// TIA Portal V19 export
DATA_BLOCK "PPrfArchive1"   // DB87
// stored: IsOnlyStoredInLoadMemory true, MemoryReserve 0
   VAR RETAIN
      PRG : Array[1.."PPRF_TOTAL_ARCHIVE_ITEMS"] of "PPrf_Data";
   END_VAR
BEGIN
   PRG[1].Header.PrgNo := 1;
   PRG[2].Header.PrgNo := 107;
   PRG[3].Header.PrgNo := 101;
   PRG[4].Header.PrgNo := 102;
   PRG[5].Header.PrgNo := 103;
   PRG[6].Header.PrgNo := 104;
   PRG[7].Header.PrgNo := 110;
   PRG[8].Header.PrgNo := 105;
   PRG[9].Header.PrgNo := 106;
   PRG[10].Header.PrgNo := 108;
   PRG[11].Header.PrgNo := 109;
   PRG[12].Header.PrgNo := 111;
   PRG[13].Header.PrgNo := 112;
   PRG[14].Header.PrgNo := 201;
   PRG[15].Header.PrgNo := 202;
   PRG[16].Header.PrgNo := 203;
   PRG[17].Header.PrgNo := 204;
   PRG[18].Header.PrgNo := 205;
   PRG[19].Header.PrgNo := 206;
   PRG[20].Header.PrgNo := 207;
   PRG[21].Header.PrgNo := 208;
   PRG[22].Header.PrgNo := 209;
   PRG[23].Header.PrgNo := 210;
   PRG[24].Header.PrgNo := 211;
   PRG[25].Header.PrgNo := 212;
   PRG[1].Header.PrgName := 'TEST';
   PRG[2].Header.PrgName := 'Semigusci G12L <S120x45x1.25>';
   PRG[3].Header.PrgName := 'Semigusci G06L <S060x40x1.25>';
   PRG[4].Header.PrgName := 'Semigusci G07L <S070x40x1.25>';
   PRG[5].Header.PrgName := 'Semigusci G08L <S080x40x1.25>';
   PRG[6].Header.PrgName := 'Semigusci G09L <S090x40x1.25>';
   PRG[7].Header.PrgName := 'Semigusci G14N <S140x45x1.5>';
   PRG[8].Header.PrgName := 'Semigusci G10L <S100x40x1.25>';
   PRG[9].Header.PrgName := 'Semigusci G11L <S110x45x1.25>';
   PRG[10].Header.PrgName := 'Semigusci G13L <S130x45x1.25>';
   PRG[11].Header.PrgName := 'Semigusci G14L <S140x45x1.25>';
   PRG[12].Header.PrgName := 'Semigusci G15N <S150x45x1.5>';
   PRG[13].Header.PrgName := 'Semigusci G18N <S180x45x1.5>';
   PRG[14].Header.PrgName := 'Accoppiato G06L <C060x40x1.25>';
   PRG[15].Header.PrgName := 'Accoppiato G07L <C070x40x1.25>';
   PRG[16].Header.PrgName := 'Accoppiato G08L <C080x40x1.25>';
   PRG[17].Header.PrgName := 'Accoppiato G09L <C090x40x1.25>';
   PRG[18].Header.PrgName := 'Accoppiato G10L <C100x40x1.25>';
   PRG[19].Header.PrgName := 'Accoppiato G11L <C110x45x1.25>';
   PRG[20].Header.PrgName := 'Accoppiato G12L <C120x45x1.25>';
   PRG[21].Header.PrgName := 'Accoppiato G13L <C130x45x1.25>';
   PRG[22].Header.PrgName := 'Accoppiato G14L <C140x45x1.25>';
   PRG[23].Header.PrgName := 'Accoppiato G14N <C140x45x1.5>';
   PRG[24].Header.PrgName := 'Accoppiato G15N <C150x45x1.5>';
   PRG[25].Header.PrgName := 'Accoppiato G18N <C180x45x1.5>';
   PRG[1..2].GeneralData.Material_Width := 220.0;
   PRG[3].GeneralData.Material_Width := 149.0;
   PRG[4].GeneralData.Material_Width := 159.0;
   PRG[5].GeneralData.Material_Width := 169.0;
   PRG[6].GeneralData.Material_Width := 179.0;
   PRG[7].GeneralData.Material_Width := 240.0;
   PRG[8].GeneralData.Material_Width := 189.0;
   PRG[9].GeneralData.Material_Width := 210.0;
   PRG[10].GeneralData.Material_Width := 230.0;
   PRG[11].GeneralData.Material_Width := 240.0;
   PRG[12].GeneralData.Material_Width := 255.0;
   PRG[13].GeneralData.Material_Width := 280.0;
   PRG[14].GeneralData.Material_Width := 149.0;
   PRG[15].GeneralData.Material_Width := 159.0;
   PRG[16].GeneralData.Material_Width := 169.0;
   PRG[17].GeneralData.Material_Width := 179.0;
   PRG[18].GeneralData.Material_Width := 189.0;
   PRG[19].GeneralData.Material_Width := 210.0;
   PRG[20].GeneralData.Material_Width := 220.0;
   PRG[21].GeneralData.Material_Width := 230.0;
   PRG[22..23].GeneralData.Material_Width := 240.0;
   PRG[24].GeneralData.Material_Width := 255.0;
   PRG[25].GeneralData.Material_Width := 280.0;
   PRG[26].GeneralData.Material_Width := 0.0;
   PRG[27].GeneralData.Material_Width := 214.0;
   PRG[28].GeneralData.Material_Width := 0.0;
   PRG[29].GeneralData.Material_Width := 236.0;
   PRG[30].GeneralData.Material_Width := 208.0;
   PRG[1].GeneralData.Material_Thickness := 0.0;
   PRG[3].GeneralData.Material_Thickness := 0.0;
   PRG[6..26].GeneralData.Material_Thickness := 0.0;
   PRG[27].GeneralData.Material_Thickness := 2.0;
   PRG[28].GeneralData.Material_Thickness := 0.0;
   PRG[29].GeneralData.Material_Thickness := 3.0;
   PRG[30].GeneralData.Material_Thickness := 1.5;
   PRG[1..25].GeneralData.Material_Tol_Min := -0.5;
   PRG[1..25].GeneralData.Material_Tol_Max := 0.5;
   PRG[14..25].GeneralData.Beam_Code := 1;
   PRG[1].GeneralData.Beam_W_A_Code := 40;
   PRG[2].GeneralData.Beam_W_A_Code := 45;
   PRG[3..6].GeneralData.Beam_W_A_Code := 40;
   PRG[7].GeneralData.Beam_W_A_Code := 45;
   PRG[8].GeneralData.Beam_W_A_Code := 40;
   PRG[9..13].GeneralData.Beam_W_A_Code := 45;
   PRG[14..18].GeneralData.Beam_W_A_Code := 40;
   PRG[19..25].GeneralData.Beam_W_A_Code := 45;
   PRG[1].GeneralData.Beam_H_B_Code := 60;
   PRG[2].GeneralData.Beam_H_B_Code := 120;
   PRG[3].GeneralData.Beam_H_B_Code := 60;
   PRG[4].GeneralData.Beam_H_B_Code := 70;
   PRG[5].GeneralData.Beam_H_B_Code := 80;
   PRG[6].GeneralData.Beam_H_B_Code := 90;
   PRG[7].GeneralData.Beam_H_B_Code := 140;
   PRG[8].GeneralData.Beam_H_B_Code := 100;
   PRG[9].GeneralData.Beam_H_B_Code := 110;
   PRG[10].GeneralData.Beam_H_B_Code := 130;
   PRG[11].GeneralData.Beam_H_B_Code := 140;
   PRG[12].GeneralData.Beam_H_B_Code := 150;
   PRG[13].GeneralData.Beam_H_B_Code := 180;
   PRG[14].GeneralData.Beam_H_B_Code := 60;
   PRG[15].GeneralData.Beam_H_B_Code := 70;
   PRG[16].GeneralData.Beam_H_B_Code := 80;
   PRG[17].GeneralData.Beam_H_B_Code := 90;
   PRG[18].GeneralData.Beam_H_B_Code := 100;
   PRG[19].GeneralData.Beam_H_B_Code := 110;
   PRG[20].GeneralData.Beam_H_B_Code := 120;
   PRG[21].GeneralData.Beam_H_B_Code := 130;
   PRG[22..23].GeneralData.Beam_H_B_Code := 140;
   PRG[24].GeneralData.Beam_H_B_Code := 150;
   PRG[25].GeneralData.Beam_H_B_Code := 180;
   PRG[1..6].GeneralData.Beam_TK_Code := 125;
   PRG[7].GeneralData.Beam_TK_Code := 150;
   PRG[8..11].GeneralData.Beam_TK_Code := 125;
   PRG[12..13].GeneralData.Beam_TK_Code := 150;
   PRG[14..22].GeneralData.Beam_TK_Code := 125;
   PRG[23..25].GeneralData.Beam_TK_Code := 150;
   PRG[1..25].GeneralData.Beam_Len_Tol_Min := -1.0;
   PRG[4..25].GeneralData.Thickness_Mark := 1;
   PRG[4..25].GeneralData.Trace_Mark := 1;
   PRG[1..2].GeneralData.PackLayout_BeamsPerLayer := 10;
   PRG[3..13].GeneralData.PackLayout_BeamsPerLayer := 0;
   PRG[14].GeneralData.PackLayout_BeamsPerLayer := 9;
   PRG[15].GeneralData.PackLayout_BeamsPerLayer := 8;
   PRG[16].GeneralData.PackLayout_BeamsPerLayer := 7;
   PRG[17..18].GeneralData.PackLayout_BeamsPerLayer := 6;
   PRG[19].GeneralData.PackLayout_BeamsPerLayer := 55;
   PRG[20].GeneralData.PackLayout_BeamsPerLayer := 5;
   PRG[21..24].GeneralData.PackLayout_BeamsPerLayer := 4;
   PRG[25].GeneralData.PackLayout_BeamsPerLayer := 3;
   PRG[1..2].GeneralData.PackLayout_Layers_Qty := 5;
   PRG[3..13].GeneralData.PackLayout_Layers_Qty := 0;
   PRG[14..25].GeneralData.PackLayout_Layers_Qty := 11;
   PRG[2].SetUp.Aut.Rollformer.Passaggio02_OP := 1.1;
   PRG[3..6].SetUp.Aut.Rollformer.Passaggio02_OP := 5.0;
   PRG[7].SetUp.Aut.Rollformer.Passaggio02_OP := 0.8;
   PRG[8].SetUp.Aut.Rollformer.Passaggio02_OP := 5.0;
   PRG[9..11].SetUp.Aut.Rollformer.Passaggio02_OP := 1.25;
   PRG[12..13].SetUp.Aut.Rollformer.Passaggio02_OP := 1.5;
   PRG[14..18].SetUp.Aut.Rollformer.Passaggio02_OP := 5.0;
   PRG[19].SetUp.Aut.Rollformer.Passaggio02_OP := 1.25;
   PRG[20].SetUp.Aut.Rollformer.Passaggio02_OP := 0.9137398;
   PRG[21].SetUp.Aut.Rollformer.Passaggio02_OP := 1.25;
   PRG[22].SetUp.Aut.Rollformer.Passaggio02_OP := 0.6;
   PRG[23].SetUp.Aut.Rollformer.Passaggio02_OP := 1.0;
   PRG[24].SetUp.Aut.Rollformer.Passaggio02_OP := 1.5;
   PRG[25].SetUp.Aut.Rollformer.Passaggio02_OP := 0.8;
   PRG[2].SetUp.Aut.Rollformer.Passaggio02_MOT := 1.1;
   PRG[3..6].SetUp.Aut.Rollformer.Passaggio02_MOT := 5.0;
   PRG[7].SetUp.Aut.Rollformer.Passaggio02_MOT := 0.8;
   PRG[8].SetUp.Aut.Rollformer.Passaggio02_MOT := 5.0;
   PRG[9..11].SetUp.Aut.Rollformer.Passaggio02_MOT := 1.25;
   PRG[12..13].SetUp.Aut.Rollformer.Passaggio02_MOT := 1.5;
   PRG[14..18].SetUp.Aut.Rollformer.Passaggio02_MOT := 5.0;
   PRG[19].SetUp.Aut.Rollformer.Passaggio02_MOT := 1.25;
   PRG[20].SetUp.Aut.Rollformer.Passaggio02_MOT := 0.9132179;
   PRG[21].SetUp.Aut.Rollformer.Passaggio02_MOT := 1.25;
   PRG[22].SetUp.Aut.Rollformer.Passaggio02_MOT := 0.6;
   PRG[23].SetUp.Aut.Rollformer.Passaggio02_MOT := 1.0;
   PRG[24].SetUp.Aut.Rollformer.Passaggio02_MOT := 1.5;
   PRG[25].SetUp.Aut.Rollformer.Passaggio02_MOT := 0.8;
   PRG[2].SetUp.Aut.Rollformer.Passaggio17_OP := 0.6;
   PRG[3..6].SetUp.Aut.Rollformer.Passaggio17_OP := 1.25;
   PRG[7].SetUp.Aut.Rollformer.Passaggio17_OP := 1.2;
   PRG[8..11].SetUp.Aut.Rollformer.Passaggio17_OP := 1.25;
   PRG[12..13].SetUp.Aut.Rollformer.Passaggio17_OP := 1.5;
   PRG[14..19].SetUp.Aut.Rollformer.Passaggio17_OP := 1.25;
   PRG[20].SetUp.Aut.Rollformer.Passaggio17_OP := 0.4124924;
   PRG[21].SetUp.Aut.Rollformer.Passaggio17_OP := 1.25;
   PRG[22].SetUp.Aut.Rollformer.Passaggio17_OP := 0.55;
   PRG[23].SetUp.Aut.Rollformer.Passaggio17_OP := 1.2;
   PRG[24].SetUp.Aut.Rollformer.Passaggio17_OP := 1.5;
   PRG[25].SetUp.Aut.Rollformer.Passaggio17_OP := 1.2;
   PRG[2].SetUp.Aut.Rollformer.Passaggio17_MOT := 0.6;
   PRG[3..6].SetUp.Aut.Rollformer.Passaggio17_MOT := 1.25;
   PRG[7].SetUp.Aut.Rollformer.Passaggio17_MOT := 1.2;
   PRG[8..11].SetUp.Aut.Rollformer.Passaggio17_MOT := 1.25;
   PRG[12..13].SetUp.Aut.Rollformer.Passaggio17_MOT := 1.5;
   PRG[14..19].SetUp.Aut.Rollformer.Passaggio17_MOT := 1.25;
   PRG[20].SetUp.Aut.Rollformer.Passaggio17_MOT := 0.9078614;
   PRG[21].SetUp.Aut.Rollformer.Passaggio17_MOT := 1.25;
   PRG[22].SetUp.Aut.Rollformer.Passaggio17_MOT := 0.55;
   PRG[23].SetUp.Aut.Rollformer.Passaggio17_MOT := 1.2;
   PRG[24].SetUp.Aut.Rollformer.Passaggio17_MOT := 1.5;
   PRG[25].SetUp.Aut.Rollformer.Passaggio17_MOT := 1.2;
   PRG[2].SetUp.Aut.Rollformer.Passaggio18_OP := 1.4;
   PRG[3..6].SetUp.Aut.Rollformer.Passaggio18_OP := 1.25;
   PRG[7].SetUp.Aut.Rollformer.Passaggio18_OP := 1.1;
   PRG[8..11].SetUp.Aut.Rollformer.Passaggio18_OP := 1.25;
   PRG[12..13].SetUp.Aut.Rollformer.Passaggio18_OP := 1.5;
   PRG[14..19].SetUp.Aut.Rollformer.Passaggio18_OP := 1.25;
   PRG[20].SetUp.Aut.Rollformer.Passaggio18_OP := 1.405658;
   PRG[21].SetUp.Aut.Rollformer.Passaggio18_OP := 1.25;
   PRG[22].SetUp.Aut.Rollformer.Passaggio18_OP := 1.4;
   PRG[23].SetUp.Aut.Rollformer.Passaggio18_OP := 1.1;
   PRG[24].SetUp.Aut.Rollformer.Passaggio18_OP := 1.5;
   PRG[25].SetUp.Aut.Rollformer.Passaggio18_OP := 1.1;
   PRG[2].SetUp.Aut.Rollformer.Passaggio18_MOT := 1.4;
   PRG[3..6].SetUp.Aut.Rollformer.Passaggio18_MOT := 1.25;
   PRG[7].SetUp.Aut.Rollformer.Passaggio18_MOT := 1.1;
   PRG[8..11].SetUp.Aut.Rollformer.Passaggio18_MOT := 1.25;
   PRG[12..13].SetUp.Aut.Rollformer.Passaggio18_MOT := 1.5;
   PRG[14..19].SetUp.Aut.Rollformer.Passaggio18_MOT := 1.25;
   PRG[20].SetUp.Aut.Rollformer.Passaggio18_MOT := 1.407493;
   PRG[21].SetUp.Aut.Rollformer.Passaggio18_MOT := 1.25;
   PRG[22].SetUp.Aut.Rollformer.Passaggio18_MOT := 1.4;
   PRG[23].SetUp.Aut.Rollformer.Passaggio18_MOT := 1.1;
   PRG[24].SetUp.Aut.Rollformer.Passaggio18_MOT := 1.5;
   PRG[25].SetUp.Aut.Rollformer.Passaggio18_MOT := 1.1;
   PRG[2].SetUp.Aut.Rollformer.Cassetta_1_OP := 101.75;
   PRG[3].SetUp.Aut.Rollformer.Cassetta_1_OP := 71.1;
   PRG[4].SetUp.Aut.Rollformer.Cassetta_1_OP := 76.1;
   PRG[5].SetUp.Aut.Rollformer.Cassetta_1_OP := 81.1;
   PRG[6].SetUp.Aut.Rollformer.Cassetta_1_OP := 86.1;
   PRG[7].SetUp.Aut.Rollformer.Cassetta_1_OP := 112.4;
   PRG[8].SetUp.Aut.Rollformer.Cassetta_1_OP := 91.1;
   PRG[9].SetUp.Aut.Rollformer.Cassetta_1_OP := 101.1;
   PRG[10].SetUp.Aut.Rollformer.Cassetta_1_OP := 111.1;
   PRG[11].SetUp.Aut.Rollformer.Cassetta_1_OP := 116.1;
   PRG[12].SetUp.Aut.Rollformer.Cassetta_1_OP := 120.0;
   PRG[13].SetUp.Aut.Rollformer.Cassetta_1_OP := 135.0;
   PRG[14].SetUp.Aut.Rollformer.Cassetta_1_OP := 71.1;
   PRG[15].SetUp.Aut.Rollformer.Cassetta_1_OP := 76.1;
   PRG[16].SetUp.Aut.Rollformer.Cassetta_1_OP := 81.1;
   PRG[17].SetUp.Aut.Rollformer.Cassetta_1_OP := 86.1;
   PRG[18].SetUp.Aut.Rollformer.Cassetta_1_OP := 91.1;
   PRG[19].SetUp.Aut.Rollformer.Cassetta_1_OP := 101.1;
   PRG[20].SetUp.Aut.Rollformer.Cassetta_1_OP := 101.7414;
   PRG[21].SetUp.Aut.Rollformer.Cassetta_1_OP := 111.1;
   PRG[22].SetUp.Aut.Rollformer.Cassetta_1_OP := 111.75;
   PRG[23].SetUp.Aut.Rollformer.Cassetta_1_OP := 112.4;
   PRG[24].SetUp.Aut.Rollformer.Cassetta_1_OP := 120.0;
   PRG[25].SetUp.Aut.Rollformer.Cassetta_1_OP := 132.4;
   PRG[2].SetUp.Aut.Rollformer.Cassetta_1_MOT := 105.5;
   PRG[3].SetUp.Aut.Rollformer.Cassetta_1_MOT := 71.2;
   PRG[4].SetUp.Aut.Rollformer.Cassetta_1_MOT := 76.2;
   PRG[5].SetUp.Aut.Rollformer.Cassetta_1_MOT := 81.2;
   PRG[6].SetUp.Aut.Rollformer.Cassetta_1_MOT := 86.2;
   PRG[7].SetUp.Aut.Rollformer.Cassetta_1_MOT := 112.1;
   PRG[8].SetUp.Aut.Rollformer.Cassetta_1_MOT := 91.2;
   PRG[9].SetUp.Aut.Rollformer.Cassetta_1_MOT := 101.2;
   PRG[10].SetUp.Aut.Rollformer.Cassetta_1_MOT := 111.2;
   PRG[11].SetUp.Aut.Rollformer.Cassetta_1_MOT := 116.2;
   PRG[12].SetUp.Aut.Rollformer.Cassetta_1_MOT := 120.0;
   PRG[13].SetUp.Aut.Rollformer.Cassetta_1_MOT := 135.0;
   PRG[14].SetUp.Aut.Rollformer.Cassetta_1_MOT := 71.2;
   PRG[15].SetUp.Aut.Rollformer.Cassetta_1_MOT := 76.2;
   PRG[16].SetUp.Aut.Rollformer.Cassetta_1_MOT := 81.2;
   PRG[17].SetUp.Aut.Rollformer.Cassetta_1_MOT := 86.2;
   PRG[18].SetUp.Aut.Rollformer.Cassetta_1_MOT := 91.2;
   PRG[19].SetUp.Aut.Rollformer.Cassetta_1_MOT := 101.2;
   PRG[20].SetUp.Aut.Rollformer.Cassetta_1_MOT := 106.4;
   PRG[21].SetUp.Aut.Rollformer.Cassetta_1_MOT := 111.2;
   PRG[22].SetUp.Aut.Rollformer.Cassetta_1_MOT := 115.8;
   PRG[23].SetUp.Aut.Rollformer.Cassetta_1_MOT := 112.1;
   PRG[24].SetUp.Aut.Rollformer.Cassetta_1_MOT := 120.0;
   PRG[25].SetUp.Aut.Rollformer.Cassetta_1_MOT := 132.1;
   PRG[2].SetUp.Aut.Rollformer.Cassetta_2_OP := 60.5;
   PRG[3].SetUp.Aut.Rollformer.Cassetta_2_OP := 30.0;
   PRG[4].SetUp.Aut.Rollformer.Cassetta_2_OP := 35.0;
   PRG[5].SetUp.Aut.Rollformer.Cassetta_2_OP := 40.0;
   PRG[6].SetUp.Aut.Rollformer.Cassetta_2_OP := 45.0;
   PRG[7].SetUp.Aut.Rollformer.Cassetta_2_OP := 70.1;
   PRG[8].SetUp.Aut.Rollformer.Cassetta_2_OP := 50.0;
   PRG[9].SetUp.Aut.Rollformer.Cassetta_2_OP := 55.0;
   PRG[10].SetUp.Aut.Rollformer.Cassetta_2_OP := 65.0;
   PRG[11].SetUp.Aut.Rollformer.Cassetta_2_OP := 70.0;
   PRG[12].SetUp.Aut.Rollformer.Cassetta_2_OP := 75.0;
   PRG[13].SetUp.Aut.Rollformer.Cassetta_2_OP := 90.0;
   PRG[14].SetUp.Aut.Rollformer.Cassetta_2_OP := 30.0;
   PRG[15].SetUp.Aut.Rollformer.Cassetta_2_OP := 35.0;
   PRG[16].SetUp.Aut.Rollformer.Cassetta_2_OP := 40.0;
   PRG[17].SetUp.Aut.Rollformer.Cassetta_2_OP := 45.0;
   PRG[18].SetUp.Aut.Rollformer.Cassetta_2_OP := 50.0;
   PRG[19].SetUp.Aut.Rollformer.Cassetta_2_OP := 55.0;
   PRG[20].SetUp.Aut.Rollformer.Cassetta_2_OP := 60.5;
   PRG[21].SetUp.Aut.Rollformer.Cassetta_2_OP := 65.0;
   PRG[22].SetUp.Aut.Rollformer.Cassetta_2_OP := 70.5;
   PRG[23].SetUp.Aut.Rollformer.Cassetta_2_OP := 69.9;
   PRG[24].SetUp.Aut.Rollformer.Cassetta_2_OP := 75.0;
   PRG[25].SetUp.Aut.Rollformer.Cassetta_2_OP := 90.1;
   PRG[2].SetUp.Aut.Rollformer.Cassetta_2_MOT := 60.35;
   PRG[3].SetUp.Aut.Rollformer.Cassetta_2_MOT := 30.25;
   PRG[4].SetUp.Aut.Rollformer.Cassetta_2_MOT := 35.25;
   PRG[5].SetUp.Aut.Rollformer.Cassetta_2_MOT := 40.25;
   PRG[6].SetUp.Aut.Rollformer.Cassetta_2_MOT := 45.25;
   PRG[7].SetUp.Aut.Rollformer.Cassetta_2_MOT := 70.5;
   PRG[8].SetUp.Aut.Rollformer.Cassetta_2_MOT := 50.25;
   PRG[9].SetUp.Aut.Rollformer.Cassetta_2_MOT := 55.25;
   PRG[10].SetUp.Aut.Rollformer.Cassetta_2_MOT := 65.25;
   PRG[11].SetUp.Aut.Rollformer.Cassetta_2_MOT := 70.25;
   PRG[12].SetUp.Aut.Rollformer.Cassetta_2_MOT := 75.0;
   PRG[13].SetUp.Aut.Rollformer.Cassetta_2_MOT := 90.0;
   PRG[14].SetUp.Aut.Rollformer.Cassetta_2_MOT := 30.25;
   PRG[15].SetUp.Aut.Rollformer.Cassetta_2_MOT := 35.25;
   PRG[16].SetUp.Aut.Rollformer.Cassetta_2_MOT := 40.25;
   PRG[17].SetUp.Aut.Rollformer.Cassetta_2_MOT := 45.25;
   PRG[18].SetUp.Aut.Rollformer.Cassetta_2_MOT := 50.25;
   PRG[19].SetUp.Aut.Rollformer.Cassetta_2_MOT := 55.25;
   PRG[20].SetUp.Aut.Rollformer.Cassetta_2_MOT := 60.00948;
   PRG[21].SetUp.Aut.Rollformer.Cassetta_2_MOT := 65.25;
   PRG[22..23].SetUp.Aut.Rollformer.Cassetta_2_MOT := 70.3;
   PRG[24].SetUp.Aut.Rollformer.Cassetta_2_MOT := 75.0;
   PRG[25].SetUp.Aut.Rollformer.Cassetta_2_MOT := 90.5;
   PRG[2].SetUp.Aut.Rollformer.Cassetta_3_OP := 59.75;
   PRG[3].SetUp.Aut.Rollformer.Cassetta_3_OP := 30.0;
   PRG[4].SetUp.Aut.Rollformer.Cassetta_3_OP := 35.0;
   PRG[5].SetUp.Aut.Rollformer.Cassetta_3_OP := 40.0;
   PRG[6].SetUp.Aut.Rollformer.Cassetta_3_OP := 45.0;
   PRG[7].SetUp.Aut.Rollformer.Cassetta_3_OP := 70.1;
   PRG[8].SetUp.Aut.Rollformer.Cassetta_3_OP := 50.0;
   PRG[9].SetUp.Aut.Rollformer.Cassetta_3_OP := 55.0;
   PRG[10].SetUp.Aut.Rollformer.Cassetta_3_OP := 65.0;
   PRG[11].SetUp.Aut.Rollformer.Cassetta_3_OP := 70.0;
   PRG[12].SetUp.Aut.Rollformer.Cassetta_3_OP := 75.0;
   PRG[13].SetUp.Aut.Rollformer.Cassetta_3_OP := 90.0;
   PRG[14].SetUp.Aut.Rollformer.Cassetta_3_OP := 30.0;
   PRG[15].SetUp.Aut.Rollformer.Cassetta_3_OP := 35.0;
   PRG[16].SetUp.Aut.Rollformer.Cassetta_3_OP := 40.0;
   PRG[17].SetUp.Aut.Rollformer.Cassetta_3_OP := 45.0;
   PRG[18].SetUp.Aut.Rollformer.Cassetta_3_OP := 50.0;
   PRG[19].SetUp.Aut.Rollformer.Cassetta_3_OP := 55.0;
   PRG[20].SetUp.Aut.Rollformer.Cassetta_3_OP := 59.74569;
   PRG[21].SetUp.Aut.Rollformer.Cassetta_3_OP := 65.0;
   PRG[22].SetUp.Aut.Rollformer.Cassetta_3_OP := 70.5;
   PRG[23].SetUp.Aut.Rollformer.Cassetta_3_OP := 69.9;
   PRG[24].SetUp.Aut.Rollformer.Cassetta_3_OP := 75.0;
   PRG[25].SetUp.Aut.Rollformer.Cassetta_3_OP := 90.1;
   PRG[2].SetUp.Aut.Rollformer.Cassetta_3_MOT := 60.5;
   PRG[3].SetUp.Aut.Rollformer.Cassetta_3_MOT := 30.25;
   PRG[4].SetUp.Aut.Rollformer.Cassetta_3_MOT := 35.25;
   PRG[5].SetUp.Aut.Rollformer.Cassetta_3_MOT := 40.25;
   PRG[6].SetUp.Aut.Rollformer.Cassetta_3_MOT := 45.25;
   PRG[7].SetUp.Aut.Rollformer.Cassetta_3_MOT := 70.5;
   PRG[8].SetUp.Aut.Rollformer.Cassetta_3_MOT := 50.25;
   PRG[9].SetUp.Aut.Rollformer.Cassetta_3_MOT := 55.25;
   PRG[10].SetUp.Aut.Rollformer.Cassetta_3_MOT := 65.25;
   PRG[11].SetUp.Aut.Rollformer.Cassetta_3_MOT := 70.25;
   PRG[12].SetUp.Aut.Rollformer.Cassetta_3_MOT := 75.0;
   PRG[13].SetUp.Aut.Rollformer.Cassetta_3_MOT := 90.0;
   PRG[14].SetUp.Aut.Rollformer.Cassetta_3_MOT := 30.25;
   PRG[15].SetUp.Aut.Rollformer.Cassetta_3_MOT := 35.25;
   PRG[16].SetUp.Aut.Rollformer.Cassetta_3_MOT := 40.25;
   PRG[17].SetUp.Aut.Rollformer.Cassetta_3_MOT := 45.25;
   PRG[18].SetUp.Aut.Rollformer.Cassetta_3_MOT := 50.25;
   PRG[19].SetUp.Aut.Rollformer.Cassetta_3_MOT := 55.25;
   PRG[20].SetUp.Aut.Rollformer.Cassetta_3_MOT := 60.00629;
   PRG[21].SetUp.Aut.Rollformer.Cassetta_3_MOT := 65.25;
   PRG[22..23].SetUp.Aut.Rollformer.Cassetta_3_MOT := 70.3;
   PRG[24].SetUp.Aut.Rollformer.Cassetta_3_MOT := 75.0;
   PRG[25].SetUp.Aut.Rollformer.Cassetta_3_MOT := 90.5;
   PRG[2].SetUp.Aut.Bordatrice.Passaggio01_L := 45.0;
   PRG[5..7].SetUp.Aut.Bordatrice.Passaggio01_L := 45.0;
   PRG[20].SetUp.Aut.Bordatrice.Passaggio01_L := 46.09322;
   PRG[22].SetUp.Aut.Bordatrice.Passaggio01_L := 46.0;
   PRG[23..24].SetUp.Aut.Bordatrice.Passaggio01_L := 45.0;
   PRG[25].SetUp.Aut.Bordatrice.Passaggio01_L := 45.5;
   PRG[2].SetUp.Aut.Bordatrice.Passaggio01_R := 45.0;
   PRG[5..7].SetUp.Aut.Bordatrice.Passaggio01_R := 45.0;
   PRG[20].SetUp.Aut.Bordatrice.Passaggio01_R := 46.09262;
   PRG[22].SetUp.Aut.Bordatrice.Passaggio01_R := 46.0;
   PRG[23..24].SetUp.Aut.Bordatrice.Passaggio01_R := 45.0;
   PRG[25].SetUp.Aut.Bordatrice.Passaggio01_R := 45.5;
   PRG[2].SetUp.Aut.Bordatrice.Passaggio02_L := 45.0;
   PRG[6].SetUp.Aut.Bordatrice.Passaggio02_L := 45.0;
   PRG[7].SetUp.Aut.Bordatrice.Passaggio02_L := 44.85;
   PRG[20].SetUp.Aut.Bordatrice.Passaggio02_L := 45.00256;
   PRG[22].SetUp.Aut.Bordatrice.Passaggio02_L := 45.0;
   PRG[23].SetUp.Aut.Bordatrice.Passaggio02_L := 44.8;
   PRG[24].SetUp.Aut.Bordatrice.Passaggio02_L := 45.0;
   PRG[25].SetUp.Aut.Bordatrice.Passaggio02_L := 44.5;
   PRG[2].SetUp.Aut.Bordatrice.Passaggio02_R := 45.0;
   PRG[6].SetUp.Aut.Bordatrice.Passaggio02_R := 45.0;
   PRG[7].SetUp.Aut.Bordatrice.Passaggio02_R := 44.85;
   PRG[20].SetUp.Aut.Bordatrice.Passaggio02_R := 45.00402;
   PRG[22].SetUp.Aut.Bordatrice.Passaggio02_R := 45.0;
   PRG[23].SetUp.Aut.Bordatrice.Passaggio02_R := 44.8;
   PRG[24].SetUp.Aut.Bordatrice.Passaggio02_R := 45.0;
   PRG[25].SetUp.Aut.Bordatrice.Passaggio02_R := 44.5;
   PRG[2].SetUp.Aut.Bordatrice.Passaggio03_L := 45.0;
   PRG[6].SetUp.Aut.Bordatrice.Passaggio03_L := 45.0;
   PRG[7].SetUp.Aut.Bordatrice.Passaggio03_L := 43.7;
   PRG[20].SetUp.Aut.Bordatrice.Passaggio03_L := 44.10418;
   PRG[22].SetUp.Aut.Bordatrice.Passaggio03_L := 45.0;
   PRG[23].SetUp.Aut.Bordatrice.Passaggio03_L := 44.0;
   PRG[24].SetUp.Aut.Bordatrice.Passaggio03_L := 45.0;
   PRG[25].SetUp.Aut.Bordatrice.Passaggio03_L := 43.7;
   PRG[2].SetUp.Aut.Bordatrice.Passaggio03_R := 45.0;
   PRG[6].SetUp.Aut.Bordatrice.Passaggio03_R := 45.0;
   PRG[7].SetUp.Aut.Bordatrice.Passaggio03_R := 43.7;
   PRG[20].SetUp.Aut.Bordatrice.Passaggio03_R := 44.49652;
   PRG[22].SetUp.Aut.Bordatrice.Passaggio03_R := 45.0;
   PRG[23].SetUp.Aut.Bordatrice.Passaggio03_R := 44.0;
   PRG[24].SetUp.Aut.Bordatrice.Passaggio03_R := 45.0;
   PRG[25].SetUp.Aut.Bordatrice.Passaggio03_R := 43.7;
   PRG[2].SetUp.Aut.Bordatrice.Passaggio04_L := 45.0;
   PRG[6].SetUp.Aut.Bordatrice.Passaggio04_L := 45.0;
   PRG[7].SetUp.Aut.Bordatrice.Passaggio04_L := 44.2;
   PRG[20].SetUp.Aut.Bordatrice.Passaggio04_L := 43.6;
   PRG[22].SetUp.Aut.Bordatrice.Passaggio04_L := 43.7;
   PRG[23].SetUp.Aut.Bordatrice.Passaggio04_L := 43.9;
   PRG[24].SetUp.Aut.Bordatrice.Passaggio04_L := 45.0;
   PRG[25].SetUp.Aut.Bordatrice.Passaggio04_L := 43.55;
   PRG[2].SetUp.Aut.Bordatrice.Passaggio04_R := 45.0;
   PRG[6].SetUp.Aut.Bordatrice.Passaggio04_R := 45.0;
   PRG[7].SetUp.Aut.Bordatrice.Passaggio04_R := 44.2;
   PRG[20].SetUp.Aut.Bordatrice.Passaggio04_R := 43.5;
   PRG[22].SetUp.Aut.Bordatrice.Passaggio04_R := 43.7;
   PRG[23].SetUp.Aut.Bordatrice.Passaggio04_R := 43.9;
   PRG[24].SetUp.Aut.Bordatrice.Passaggio04_R := 45.0;
   PRG[25].SetUp.Aut.Bordatrice.Passaggio04_R := 43.55;
   PRG[7].SetUp.Aut.Bordatrice.Cassetta_1_OP := 141.0;
   PRG[20].SetUp.Aut.Bordatrice.Cassetta_1_OP := 119.8;
   PRG[22].SetUp.Aut.Bordatrice.Cassetta_1_OP := 139.7;
   PRG[23].SetUp.Aut.Bordatrice.Cassetta_1_OP := 140.5;
   PRG[25].SetUp.Aut.Bordatrice.Cassetta_1_OP := 180.1;
   PRG[2].SetUp.Man.X[15] := 109.3;
   PRG[2].SetUp.Man.X[16] := 111.3;
   PRG[2].SetUp.Man.X[17] := 7.6;
   PRG[2].SetUp.Man.X[18] := 9.5;
   PRG[2].SetUp.Man.X[19] := 7.6;
   PRG[2].SetUp.Man.X[20] := 9.5;
   PRG[2].SetUp.Man.X[21] := 45.1;
   PRG[2].SetUp.Man.X[22] := 43.5;
   PRG[2].SetUp.Man.X[23] := 45.1;
   PRG[2].SetUp.Man.X[24] := 43.5;
   PRG[2].SetUp.Man.X[25] := 45.1;
   PRG[2].SetUp.Man.X[26] := 43.5;
   PRG[2].SetUp.Man.X[27] := 0.1;
   PRG[2].SetUp.Man.X[28] := 87.6;
   PRG[2].SetUp.Man.X[29] := 84.8;
   PRG[2].SetUp.Man.X[30] := 58.75;
   PRG[2].SetUp.Man.X[31] := 60.0;
   PRG[2].SetUp.Man.X[32] := 58.75;
   PRG[2].SetUp.Man.X[33] := 60.0;
   PRG[3].SetUp.Man.X[15] := 77.6;
   PRG[3].SetUp.Man.X[16] := 71.9;
   PRG[3].SetUp.Man.X[17] := 8.4;
   PRG[3].SetUp.Man.X[18] := 7.0;
   PRG[3].SetUp.Man.X[19] := 8.4;
   PRG[3].SetUp.Man.X[20] := 7.0;
   PRG[3].SetUp.Man.X[21] := 40.1;
   PRG[3].SetUp.Man.X[22] := 38.5;
   PRG[3].SetUp.Man.X[23] := 40.1;
   PRG[3].SetUp.Man.X[24] := 38.5;
   PRG[3].SetUp.Man.X[25] := 40.1;
   PRG[3].SetUp.Man.X[26] := 38.5;
   PRG[3].SetUp.Man.X[27] := 1.0;
   PRG[3].SetUp.Man.X[28] := 87.0;
   PRG[3].SetUp.Man.X[29] := 84.2;
   PRG[3].SetUp.Man.X[30] := 28.75;
   PRG[3].SetUp.Man.X[31] := 30.0;
   PRG[3].SetUp.Man.X[32] := 28.75;
   PRG[3].SetUp.Man.X[33] := 30.0;
   PRG[4].SetUp.Man.X[15] := 82.5;
   PRG[4].SetUp.Man.X[16] := 79.5;
   PRG[4].SetUp.Man.X[17] := 9.75;
   PRG[4].SetUp.Man.X[18] := 5.8;
   PRG[4].SetUp.Man.X[19] := 9.75;
   PRG[4].SetUp.Man.X[20] := 5.8;
   PRG[4].SetUp.Man.X[21] := 41.1;
   PRG[4].SetUp.Man.X[22] := 41.2;
   PRG[4].SetUp.Man.X[23] := 41.1;
   PRG[4].SetUp.Man.X[24] := 41.2;
   PRG[4].SetUp.Man.X[25] := 41.1;
   PRG[4].SetUp.Man.X[26] := 41.2;
   PRG[4].SetUp.Man.X[27] := -0.4;
   PRG[4].SetUp.Man.X[30] := 35.0;
   PRG[4].SetUp.Man.X[31] := 33.75;
   PRG[4].SetUp.Man.X[32] := 35.0;
   PRG[4].SetUp.Man.X[33] := 33.75;
   PRG[5].SetUp.Man.X[15] := 87.5;
   PRG[5].SetUp.Man.X[16] := 84.5;
   PRG[5].SetUp.Man.X[17] := 9.75;
   PRG[5].SetUp.Man.X[18] := 5.8;
   PRG[5].SetUp.Man.X[19] := 9.75;
   PRG[5].SetUp.Man.X[20] := 5.8;
   PRG[5].SetUp.Man.X[21] := 41.1;
   PRG[5].SetUp.Man.X[22] := 41.2;
   PRG[5].SetUp.Man.X[23] := 41.1;
   PRG[5].SetUp.Man.X[24] := 41.2;
   PRG[5].SetUp.Man.X[25] := 41.1;
   PRG[5].SetUp.Man.X[26] := 41.2;
   PRG[5].SetUp.Man.X[27] := -0.4;
   PRG[5].SetUp.Man.X[30] := 38.75;
   PRG[5].SetUp.Man.X[31] := 40.0;
   PRG[5].SetUp.Man.X[32] := 38.75;
   PRG[5].SetUp.Man.X[33] := 40.0;
   PRG[6].SetUp.Man.X[15] := 92.5;
   PRG[6].SetUp.Man.X[16] := 89.5;
   PRG[6].SetUp.Man.X[17] := 9.75;
   PRG[6].SetUp.Man.X[18] := 5.8;
   PRG[6].SetUp.Man.X[19] := 9.75;
   PRG[6].SetUp.Man.X[20] := 5.8;
   PRG[6].SetUp.Man.X[21] := 41.1;
   PRG[6].SetUp.Man.X[22] := 41.2;
   PRG[6].SetUp.Man.X[23] := 41.1;
   PRG[6].SetUp.Man.X[24] := 41.2;
   PRG[6].SetUp.Man.X[25] := 41.1;
   PRG[6].SetUp.Man.X[26] := 41.2;
   PRG[6].SetUp.Man.X[27] := -0.4;
   PRG[6].SetUp.Man.X[30] := 43.8;
   PRG[6].SetUp.Man.X[31] := 45.0;
   PRG[6].SetUp.Man.X[32] := 43.8;
   PRG[6].SetUp.Man.X[33] := 45.0;
   PRG[7].SetUp.Man.X[15..16] := 122.5;
   PRG[7].SetUp.Man.X[17..20] := 10.0;
   PRG[7].SetUp.Man.X[21..26] := 45.0;
   PRG[7].SetUp.Man.X[30] := 68.5;
   PRG[7].SetUp.Man.X[31] := 70.0;
   PRG[7].SetUp.Man.X[32] := 68.5;
   PRG[7].SetUp.Man.X[33] := 70.0;
   PRG[8].SetUp.Man.X[15] := 97.5;
   PRG[8].SetUp.Man.X[16] := 94.5;
   PRG[8].SetUp.Man.X[17] := 9.75;
   PRG[8].SetUp.Man.X[18] := 5.8;
   PRG[8].SetUp.Man.X[19] := 9.75;
   PRG[8].SetUp.Man.X[20] := 5.8;
   PRG[8].SetUp.Man.X[21] := 41.1;
   PRG[8].SetUp.Man.X[22] := 41.2;
   PRG[8].SetUp.Man.X[23] := 41.1;
   PRG[8].SetUp.Man.X[24] := 41.2;
   PRG[8].SetUp.Man.X[25] := 41.1;
   PRG[8].SetUp.Man.X[26] := 41.2;
   PRG[8].SetUp.Man.X[27] := -0.4;
   PRG[8].SetUp.Man.X[30] := 48.8;
   PRG[8].SetUp.Man.X[31] := 50.0;
   PRG[8].SetUp.Man.X[32] := 48.8;
   PRG[8].SetUp.Man.X[33] := 50.0;
   PRG[9].SetUp.Man.X[15] := 97.5;
   PRG[9].SetUp.Man.X[16] := 94.5;
   PRG[9].SetUp.Man.X[17] := 9.75;
   PRG[9].SetUp.Man.X[18] := 5.8;
   PRG[9].SetUp.Man.X[19] := 9.75;
   PRG[9].SetUp.Man.X[20] := 5.8;
   PRG[9].SetUp.Man.X[21] := 46.1;
   PRG[9].SetUp.Man.X[22] := 46.2;
   PRG[9].SetUp.Man.X[23] := 46.1;
   PRG[9].SetUp.Man.X[24] := 46.2;
   PRG[9].SetUp.Man.X[25] := 46.1;
   PRG[9].SetUp.Man.X[26] := 46.2;
   PRG[9].SetUp.Man.X[27] := -0.4;
   PRG[9].SetUp.Man.X[30] := 53.8;
   PRG[9].SetUp.Man.X[31] := 55.0;
   PRG[9].SetUp.Man.X[32] := 53.8;
   PRG[9].SetUp.Man.X[33] := 55.0;
   PRG[10].SetUp.Man.X[15] := 118.0;
   PRG[10].SetUp.Man.X[16] := 115.0;
   PRG[10].SetUp.Man.X[17] := 9.75;
   PRG[10].SetUp.Man.X[18] := 5.8;
   PRG[10].SetUp.Man.X[19] := 9.8;
   PRG[10].SetUp.Man.X[20] := 5.8;
   PRG[10].SetUp.Man.X[21] := 46.1;
   PRG[10].SetUp.Man.X[22] := 46.2;
   PRG[10].SetUp.Man.X[23] := 46.1;
   PRG[10].SetUp.Man.X[24] := 46.2;
   PRG[10].SetUp.Man.X[25] := 46.1;
   PRG[10].SetUp.Man.X[26] := 46.2;
   PRG[10].SetUp.Man.X[27] := -0.4;
   PRG[10].SetUp.Man.X[30] := 63.75;
   PRG[10].SetUp.Man.X[31] := 65.0;
   PRG[10].SetUp.Man.X[32] := 63.75;
   PRG[10].SetUp.Man.X[33] := 65.0;
   PRG[11].SetUp.Man.X[15] := 123.0;
   PRG[11].SetUp.Man.X[16] := 120.0;
   PRG[11].SetUp.Man.X[17] := 7.6;
   PRG[11].SetUp.Man.X[18] := 9.5;
   PRG[11].SetUp.Man.X[19] := 7.6;
   PRG[11].SetUp.Man.X[20] := 9.5;
   PRG[11].SetUp.Man.X[21] := 46.1;
   PRG[11].SetUp.Man.X[22] := 46.2;
   PRG[11].SetUp.Man.X[23] := 46.1;
   PRG[11].SetUp.Man.X[24] := 46.2;
   PRG[11].SetUp.Man.X[25] := 46.1;
   PRG[11].SetUp.Man.X[26] := 46.2;
   PRG[11].SetUp.Man.X[27] := -0.4;
   PRG[11].SetUp.Man.X[30] := 68.8;
   PRG[11].SetUp.Man.X[31] := 70.0;
   PRG[11].SetUp.Man.X[32] := 68.8;
   PRG[11].SetUp.Man.X[33] := 70.0;
   PRG[12].SetUp.Man.X[15] := 126.5;
   PRG[12].SetUp.Man.X[16] := 124.8;
   PRG[12].SetUp.Man.X[17] := 9.0;
   PRG[12].SetUp.Man.X[18] := 12.25;
   PRG[12].SetUp.Man.X[19] := 9.0;
   PRG[12].SetUp.Man.X[20] := 12.25;
   PRG[12].SetUp.Man.X[21] := 42.5;
   PRG[12].SetUp.Man.X[22] := 42.4;
   PRG[12].SetUp.Man.X[23] := 42.5;
   PRG[12].SetUp.Man.X[24] := 42.4;
   PRG[12].SetUp.Man.X[25] := 42.5;
   PRG[12].SetUp.Man.X[26] := 42.4;
   PRG[12].SetUp.Man.X[27] := 0.1;
   PRG[12].SetUp.Man.X[28] := 86.7;
   PRG[12].SetUp.Man.X[29] := 84.0;
   PRG[12].SetUp.Man.X[30] := 73.5;
   PRG[12].SetUp.Man.X[31] := 75.0;
   PRG[12].SetUp.Man.X[32] := 73.5;
   PRG[12].SetUp.Man.X[33] := 75.0;
   PRG[13].SetUp.Man.X[15..16] := 142.5;
   PRG[13].SetUp.Man.X[17..20] := 10.0;
   PRG[13].SetUp.Man.X[21..26] := 45.0;
   PRG[13].SetUp.Man.X[30] := 88.5;
   PRG[13].SetUp.Man.X[31] := 90.0;
   PRG[13].SetUp.Man.X[32] := 88.5;
   PRG[13].SetUp.Man.X[33] := 90.0;
   PRG[14].SetUp.Man.X[15] := 77.6;
   PRG[14].SetUp.Man.X[16] := 71.9;
   PRG[14].SetUp.Man.X[17] := 8.4;
   PRG[14].SetUp.Man.X[18] := 7.0;
   PRG[14].SetUp.Man.X[19] := 8.4;
   PRG[14].SetUp.Man.X[20] := 7.0;
   PRG[14].SetUp.Man.X[21] := 40.1;
   PRG[14].SetUp.Man.X[22] := 38.5;
   PRG[14].SetUp.Man.X[23] := 40.1;
   PRG[14].SetUp.Man.X[24] := 38.5;
   PRG[14].SetUp.Man.X[25] := 40.1;
   PRG[14].SetUp.Man.X[26] := 38.5;
   PRG[14].SetUp.Man.X[27] := 1.0;
   PRG[14].SetUp.Man.X[28] := 87.0;
   PRG[14].SetUp.Man.X[29] := 84.2;
   PRG[14].SetUp.Man.X[30] := 28.75;
   PRG[14].SetUp.Man.X[31] := 30.0;
   PRG[14].SetUp.Man.X[32] := 28.75;
   PRG[14].SetUp.Man.X[33] := 30.0;
   PRG[15].SetUp.Man.X[15] := 82.5;
   PRG[15].SetUp.Man.X[16] := 79.5;
   PRG[15].SetUp.Man.X[17] := 9.75;
   PRG[15].SetUp.Man.X[18] := 5.8;
   PRG[15].SetUp.Man.X[19] := 9.75;
   PRG[15].SetUp.Man.X[20] := 5.8;
   PRG[15].SetUp.Man.X[21] := 41.1;
   PRG[15].SetUp.Man.X[22] := 41.2;
   PRG[15].SetUp.Man.X[23] := 41.1;
   PRG[15].SetUp.Man.X[24] := 41.2;
   PRG[15].SetUp.Man.X[25] := 41.1;
   PRG[15].SetUp.Man.X[26] := 41.2;
   PRG[15].SetUp.Man.X[27] := -0.4;
   PRG[15].SetUp.Man.X[30] := 35.0;
   PRG[15].SetUp.Man.X[31] := 33.75;
   PRG[15].SetUp.Man.X[32] := 35.0;
   PRG[15].SetUp.Man.X[33] := 33.75;
   PRG[16].SetUp.Man.X[15] := 87.5;
   PRG[16].SetUp.Man.X[16] := 84.5;
   PRG[16].SetUp.Man.X[17] := 9.75;
   PRG[16].SetUp.Man.X[18] := 5.8;
   PRG[16].SetUp.Man.X[19] := 9.75;
   PRG[16].SetUp.Man.X[20] := 5.8;
   PRG[16].SetUp.Man.X[21] := 41.1;
   PRG[16].SetUp.Man.X[22] := 41.2;
   PRG[16].SetUp.Man.X[23] := 41.1;
   PRG[16].SetUp.Man.X[24] := 41.2;
   PRG[16].SetUp.Man.X[25] := 41.1;
   PRG[16].SetUp.Man.X[26] := 41.2;
   PRG[16].SetUp.Man.X[27] := -0.4;
   PRG[16].SetUp.Man.X[30] := 38.75;
   PRG[16].SetUp.Man.X[31] := 40.0;
   PRG[16].SetUp.Man.X[32] := 38.75;
   PRG[16].SetUp.Man.X[33] := 40.0;
   PRG[17].SetUp.Man.X[15] := 92.5;
   PRG[17].SetUp.Man.X[16] := 89.5;
   PRG[17].SetUp.Man.X[17] := 9.75;
   PRG[17].SetUp.Man.X[18] := 5.8;
   PRG[17].SetUp.Man.X[19] := 9.75;
   PRG[17].SetUp.Man.X[20] := 5.8;
   PRG[17].SetUp.Man.X[21] := 41.1;
   PRG[17].SetUp.Man.X[22] := 41.2;
   PRG[17].SetUp.Man.X[23] := 41.1;
   PRG[17].SetUp.Man.X[24] := 41.2;
   PRG[17].SetUp.Man.X[25] := 41.1;
   PRG[17].SetUp.Man.X[26] := 41.2;
   PRG[17].SetUp.Man.X[27] := -0.4;
   PRG[17].SetUp.Man.X[30] := 43.8;
   PRG[17].SetUp.Man.X[31] := 45.0;
   PRG[17].SetUp.Man.X[32] := 43.8;
   PRG[17].SetUp.Man.X[33] := 45.0;
   PRG[18].SetUp.Man.X[15] := 97.5;
   PRG[18].SetUp.Man.X[16] := 94.5;
   PRG[18].SetUp.Man.X[17] := 9.75;
   PRG[18].SetUp.Man.X[18] := 5.8;
   PRG[18].SetUp.Man.X[19] := 9.75;
   PRG[18].SetUp.Man.X[20] := 5.8;
   PRG[18].SetUp.Man.X[21] := 41.1;
   PRG[18].SetUp.Man.X[22] := 41.2;
   PRG[18].SetUp.Man.X[23] := 41.1;
   PRG[18].SetUp.Man.X[24] := 41.2;
   PRG[18].SetUp.Man.X[25] := 41.1;
   PRG[18].SetUp.Man.X[26] := 41.2;
   PRG[18].SetUp.Man.X[27] := -0.4;
   PRG[18].SetUp.Man.X[30] := 48.8;
   PRG[18].SetUp.Man.X[31] := 50.0;
   PRG[18].SetUp.Man.X[32] := 48.8;
   PRG[18].SetUp.Man.X[33] := 50.0;
   PRG[19].SetUp.Man.X[15] := 97.5;
   PRG[19].SetUp.Man.X[16] := 94.5;
   PRG[19].SetUp.Man.X[17] := 9.75;
   PRG[19].SetUp.Man.X[18] := 5.8;
   PRG[19].SetUp.Man.X[19] := 9.75;
   PRG[19].SetUp.Man.X[20] := 5.8;
   PRG[19].SetUp.Man.X[21] := 46.1;
   PRG[19].SetUp.Man.X[22] := 46.2;
   PRG[19].SetUp.Man.X[23] := 46.1;
   PRG[19].SetUp.Man.X[24] := 46.2;
   PRG[19].SetUp.Man.X[25] := 46.1;
   PRG[19].SetUp.Man.X[26] := 46.2;
   PRG[19].SetUp.Man.X[27] := -0.4;
   PRG[19].SetUp.Man.X[30] := 53.8;
   PRG[19].SetUp.Man.X[31] := 55.0;
   PRG[19].SetUp.Man.X[32] := 53.8;
   PRG[19].SetUp.Man.X[33] := 55.0;
   PRG[20].SetUp.Man.X[15] := 109.3;
   PRG[20].SetUp.Man.X[16] := 111.3;
   PRG[20].SetUp.Man.X[17] := 7.6;
   PRG[20].SetUp.Man.X[18] := 9.5;
   PRG[20].SetUp.Man.X[19] := 7.6;
   PRG[20].SetUp.Man.X[20] := 9.5;
   PRG[20].SetUp.Man.X[21] := 45.1;
   PRG[20].SetUp.Man.X[22] := 43.5;
   PRG[20].SetUp.Man.X[23] := 45.1;
   PRG[20].SetUp.Man.X[24] := 43.5;
   PRG[20].SetUp.Man.X[25] := 45.1;
   PRG[20].SetUp.Man.X[26] := 43.5;
   PRG[20].SetUp.Man.X[27] := 0.1;
   PRG[20].SetUp.Man.X[28] := 87.6;
   PRG[20].SetUp.Man.X[29] := 84.8;
   PRG[20].SetUp.Man.X[30] := 58.75;
   PRG[20].SetUp.Man.X[31] := 60.0;
   PRG[20].SetUp.Man.X[32] := 58.75;
   PRG[20].SetUp.Man.X[33] := 60.0;
   PRG[21].SetUp.Man.X[15] := 118.0;
   PRG[21].SetUp.Man.X[16] := 115.0;
   PRG[21].SetUp.Man.X[17] := 9.75;
   PRG[21].SetUp.Man.X[18] := 5.8;
   PRG[21].SetUp.Man.X[19] := 9.8;
   PRG[21].SetUp.Man.X[20] := 5.8;
   PRG[21].SetUp.Man.X[21] := 46.1;
   PRG[21].SetUp.Man.X[22] := 46.2;
   PRG[21].SetUp.Man.X[23] := 46.1;
   PRG[21].SetUp.Man.X[24] := 46.2;
   PRG[21].SetUp.Man.X[25] := 46.1;
   PRG[21].SetUp.Man.X[26] := 46.2;
   PRG[21].SetUp.Man.X[27] := -0.4;
   PRG[21].SetUp.Man.X[30] := 63.75;
   PRG[21].SetUp.Man.X[31] := 65.0;
   PRG[21].SetUp.Man.X[32] := 63.75;
   PRG[21].SetUp.Man.X[33] := 65.0;
   PRG[22].SetUp.Man.X[15] := 123.0;
   PRG[22].SetUp.Man.X[16] := 120.0;
   PRG[22].SetUp.Man.X[17] := 7.6;
   PRG[22].SetUp.Man.X[18] := 9.5;
   PRG[22].SetUp.Man.X[19] := 7.6;
   PRG[22].SetUp.Man.X[20] := 9.5;
   PRG[22].SetUp.Man.X[21] := 46.1;
   PRG[22].SetUp.Man.X[22] := 46.2;
   PRG[22].SetUp.Man.X[23] := 46.1;
   PRG[22].SetUp.Man.X[24] := 46.2;
   PRG[22].SetUp.Man.X[25] := 46.1;
   PRG[22].SetUp.Man.X[26] := 46.2;
   PRG[22].SetUp.Man.X[27] := -0.4;
   PRG[22].SetUp.Man.X[30] := 68.8;
   PRG[22].SetUp.Man.X[31] := 70.0;
   PRG[22].SetUp.Man.X[32] := 68.8;
   PRG[22].SetUp.Man.X[33] := 70.0;
   PRG[23].SetUp.Man.X[15..16] := 122.5;
   PRG[23].SetUp.Man.X[17..20] := 10.0;
   PRG[23].SetUp.Man.X[21..26] := 45.0;
   PRG[23].SetUp.Man.X[30] := 68.5;
   PRG[23].SetUp.Man.X[31] := 70.0;
   PRG[23].SetUp.Man.X[32] := 68.5;
   PRG[23].SetUp.Man.X[33] := 70.0;
   PRG[24].SetUp.Man.X[15] := 126.5;
   PRG[24].SetUp.Man.X[16] := 124.8;
   PRG[24].SetUp.Man.X[17] := 9.0;
   PRG[24].SetUp.Man.X[18] := 12.25;
   PRG[24].SetUp.Man.X[19] := 9.0;
   PRG[24].SetUp.Man.X[20] := 12.25;
   PRG[24].SetUp.Man.X[21] := 42.5;
   PRG[24].SetUp.Man.X[22] := 42.4;
   PRG[24].SetUp.Man.X[23] := 42.5;
   PRG[24].SetUp.Man.X[24] := 42.4;
   PRG[24].SetUp.Man.X[25] := 42.5;
   PRG[24].SetUp.Man.X[26] := 42.4;
   PRG[24].SetUp.Man.X[27] := 0.1;
   PRG[24].SetUp.Man.X[28] := 86.7;
   PRG[24].SetUp.Man.X[29] := 84.0;
   PRG[24].SetUp.Man.X[30] := 73.5;
   PRG[24].SetUp.Man.X[31] := 75.0;
   PRG[24].SetUp.Man.X[32] := 73.5;
   PRG[24].SetUp.Man.X[33] := 75.0;
   PRG[25].SetUp.Man.X[15..16] := 142.5;
   PRG[25].SetUp.Man.X[17..20] := 10.0;
   PRG[25].SetUp.Man.X[21..26] := 45.0;
   PRG[25].SetUp.Man.X[30] := 88.5;
   PRG[25].SetUp.Man.X[31] := 90.0;
   PRG[25].SetUp.Man.X[32] := 88.5;
   PRG[25].SetUp.Man.X[33] := 90.0;
   PRG[2].SetUp.Man.Y[1..2] := 120;
   PRG[3].SetUp.Man.Y[1..2] := 60;
   PRG[4].SetUp.Man.Y[1..2] := 70;
   PRG[5].SetUp.Man.Y[1..2] := 80;
   PRG[6].SetUp.Man.Y[1..2] := 90;
   PRG[7].SetUp.Man.Y[1..2] := 140;
   PRG[8].SetUp.Man.Y[1..2] := 100;
   PRG[9].SetUp.Man.Y[1..2] := 110;
   PRG[10].SetUp.Man.Y[1..2] := 130;
   PRG[11].SetUp.Man.Y[1..2] := 140;
   PRG[12].SetUp.Man.Y[1..2] := 150;
   PRG[13].SetUp.Man.Y[1..2] := 180;
   PRG[14].SetUp.Man.Y[1..2] := 60;
   PRG[15].SetUp.Man.Y[1..2] := 70;
   PRG[16].SetUp.Man.Y[1..2] := 80;
   PRG[17].SetUp.Man.Y[1..2] := 90;
   PRG[18].SetUp.Man.Y[1..2] := 100;
   PRG[19].SetUp.Man.Y[1..2] := 110;
   PRG[20].SetUp.Man.Y[1..2] := 120;
   PRG[21].SetUp.Man.Y[1..2] := 130;
   PRG[22].SetUp.Man.Y[1..2] := 140;
   PRG[23].SetUp.Man.Y[1..2] := 140;
   PRG[24].SetUp.Man.Y[1..2] := 150;
   PRG[25].SetUp.Man.Y[1..2] := 180;
   PRG[1..2].A01_CoilHandling.MaterialFeeding.DecoilerFeedMode := 3;
   PRG[3..25].A01_CoilHandling.MaterialFeeding.DecoilerFeedMode := 1;
   PRG[26].A01_CoilHandling.MaterialFeeding.DecoilerFeedMode := 0;
   PRG[27].A01_CoilHandling.MaterialFeeding.DecoilerFeedMode := 1;
   PRG[28].A01_CoilHandling.MaterialFeeding.DecoilerFeedMode := 0;
   PRG[29..30].A01_CoilHandling.MaterialFeeding.DecoilerFeedMode := 1;
   PRG[1..2].A01_CoilHandling.MaterialFeeding.StraightenerRollsUse := 0;
   PRG[3..25].A01_CoilHandling.MaterialFeeding.StraightenerRollsUse := 1;
   PRG[26].A01_CoilHandling.MaterialFeeding.StraightenerRollsUse := 0;
   PRG[27].A01_CoilHandling.MaterialFeeding.StraightenerRollsUse := 3;
   PRG[28].A01_CoilHandling.MaterialFeeding.StraightenerRollsUse := 0;
   PRG[29..30].A01_CoilHandling.MaterialFeeding.StraightenerRollsUse := 3;
   PRG[1..19].A01_CoilHandling.MaterialFeeding.Vel := 5000.0;
   PRG[20].A01_CoilHandling.MaterialFeeding.Vel := 8000.0;
   PRG[21..25].A01_CoilHandling.MaterialFeeding.Vel := 5000.0;
   PRG[26].A01_CoilHandling.MaterialFeeding.Vel := 0.0;
   PRG[27].A01_CoilHandling.MaterialFeeding.Vel := 10000.0;
   PRG[28].A01_CoilHandling.MaterialFeeding.Vel := 0.0;
   PRG[29..30].A01_CoilHandling.MaterialFeeding.Vel := 10000.0;
   PRG[1..25].A01_CoilHandling.MaterialFeeding.Acc := 1000.0;
   PRG[26].A01_CoilHandling.MaterialFeeding.Acc := 0.0;
   PRG[27].A01_CoilHandling.MaterialFeeding.Acc := 500.0;
   PRG[28].A01_CoilHandling.MaterialFeeding.Acc := 0.0;
   PRG[29..30].A01_CoilHandling.MaterialFeeding.Acc := 500.0;
   PRG[1..25].A01_CoilHandling.MaterialFeeding.Dec := 1000.0;
   PRG[26].A01_CoilHandling.MaterialFeeding.Dec := 0.0;
   PRG[27].A01_CoilHandling.MaterialFeeding.Dec := 1000.0;
   PRG[28].A01_CoilHandling.MaterialFeeding.Dec := 0.0;
   PRG[29..30].A01_CoilHandling.MaterialFeeding.Dec := 1000.0;
   PRG[1..25].A01_CoilHandling.MaterialFeeding.Jerk := 10000.0;
   PRG[26].A01_CoilHandling.MaterialFeeding.Jerk := 0.0;
   PRG[27].A01_CoilHandling.MaterialFeeding.Jerk := 1000.0;
   PRG[28].A01_CoilHandling.MaterialFeeding.Jerk := 0.0;
   PRG[29..30].A01_CoilHandling.MaterialFeeding.Jerk := 1000.0;
   PRG[1..6].A01_CoilHandling.WeldingCycle.MeasureSheetEdgeReference := 300.0;
   PRG[7].A01_CoilHandling.WeldingCycle.MeasureSheetEdgeReference := 284.0;
   PRG[8..25].A01_CoilHandling.WeldingCycle.MeasureSheetEdgeReference := 300.0;
   PRG[26].A01_CoilHandling.WeldingCycle.MeasureSheetEdgeReference := 0.0;
   PRG[27].A01_CoilHandling.WeldingCycle.MeasureSheetEdgeReference := 443.0;
   PRG[28].A01_CoilHandling.WeldingCycle.MeasureSheetEdgeReference := 0.0;
   PRG[29..30].A01_CoilHandling.WeldingCycle.MeasureSheetEdgeReference := 443.0;
   PRG[1..25].A01_CoilHandling.WeldingCycle.CorrStartWelding := 1.0;
   PRG[1..25].A01_CoilHandling.WeldingCycle.CorrStopWelding := -1.0;
   PRG[1..26].A02_1_PartsCutting.Rollformer.Code := 0;
   PRG[27].A02_1_PartsCutting.Rollformer.Code := 1;
   PRG[28].A02_1_PartsCutting.Rollformer.Code := 0;
   PRG[29..30].A02_1_PartsCutting.Rollformer.Code := 1;
   PRG[1].A02_1_PartsCutting.Rollformer.FAK := 0.0;
   PRG[2..21].A02_1_PartsCutting.Rollformer.FAK := 1.0;
   PRG[22..23].A02_1_PartsCutting.Rollformer.FAK := 1.0003;
   PRG[24..25].A02_1_PartsCutting.Rollformer.FAK := 1.0;
   PRG[26].A02_1_PartsCutting.Rollformer.FAK := 0.0;
   PRG[27].A02_1_PartsCutting.Rollformer.FAK := 1.0;
   PRG[28].A02_1_PartsCutting.Rollformer.FAK := 0.0;
   PRG[29..30].A02_1_PartsCutting.Rollformer.FAK := 1.0;
   PRG[1].A02_1_PartsCutting.Rollformer.Acc := 0.0;
   PRG[2..25].A02_1_PartsCutting.Rollformer.Acc := 500.0;
   PRG[26].A02_1_PartsCutting.Rollformer.Acc := 0.0;
   PRG[27].A02_1_PartsCutting.Rollformer.Acc := 500.0;
   PRG[28].A02_1_PartsCutting.Rollformer.Acc := 0.0;
   PRG[29..30].A02_1_PartsCutting.Rollformer.Acc := 500.0;
   PRG[1].A02_1_PartsCutting.Rollformer.Dec := 0.0;
   PRG[2..25].A02_1_PartsCutting.Rollformer.Dec := 500.0;
   PRG[26].A02_1_PartsCutting.Rollformer.Dec := 0.0;
   PRG[27].A02_1_PartsCutting.Rollformer.Dec := 500.0;
   PRG[28].A02_1_PartsCutting.Rollformer.Dec := 0.0;
   PRG[29..30].A02_1_PartsCutting.Rollformer.Dec := 500.0;
   PRG[1].A02_1_PartsCutting.Rollformer.Jerk := 0.0;
   PRG[2..25].A02_1_PartsCutting.Rollformer.Jerk := 5000.0;
   PRG[26].A02_1_PartsCutting.Rollformer.Jerk := 0.0;
   PRG[27].A02_1_PartsCutting.Rollformer.Jerk := 10000.0;
   PRG[28].A02_1_PartsCutting.Rollformer.Jerk := 0.0;
   PRG[29..30].A02_1_PartsCutting.Rollformer.Jerk := 10000.0;
   PRG[1].A02_1_PartsCutting.Rollformer.TAxConfig.EncoderInverseDirection := FALSE;
   PRG[12].A02_1_PartsCutting.Rollformer.TAxConfig.EncoderInverseDirection := FALSE;
   PRG[1].A02_1_PartsCutting.Rollformer.TAxConfig.LoadGearNumerator := 0;
   PRG[2..25].A02_1_PartsCutting.Rollformer.TAxConfig.LoadGearNumerator := 37895;
   PRG[26].A02_1_PartsCutting.Rollformer.TAxConfig.LoadGearNumerator := 0;
   PRG[27].A02_1_PartsCutting.Rollformer.TAxConfig.LoadGearNumerator := 37895;
   PRG[28].A02_1_PartsCutting.Rollformer.TAxConfig.LoadGearNumerator := 0;
   PRG[29..30].A02_1_PartsCutting.Rollformer.TAxConfig.LoadGearNumerator := 37895;
   PRG[1].A02_1_PartsCutting.Rollformer.TAxConfig.LoadGearDenominator := 0;
   PRG[2..25].A02_1_PartsCutting.Rollformer.TAxConfig.LoadGearDenominator := 1000;
   PRG[26].A02_1_PartsCutting.Rollformer.TAxConfig.LoadGearDenominator := 0;
   PRG[27].A02_1_PartsCutting.Rollformer.TAxConfig.LoadGearDenominator := 1000;
   PRG[28].A02_1_PartsCutting.Rollformer.TAxConfig.LoadGearDenominator := 0;
   PRG[29..30].A02_1_PartsCutting.Rollformer.TAxConfig.LoadGearDenominator := 1000;
   PRG[1].A02_1_PartsCutting.Rollformer.TAxConfig.MechanicsLeadScrew := 0.0;
   PRG[2..25].A02_1_PartsCutting.Rollformer.TAxConfig.MechanicsLeadScrew := 622.0;
   PRG[26].A02_1_PartsCutting.Rollformer.TAxConfig.MechanicsLeadScrew := 0.0;
   PRG[27].A02_1_PartsCutting.Rollformer.TAxConfig.MechanicsLeadScrew := 622.0;
   PRG[28].A02_1_PartsCutting.Rollformer.TAxConfig.MechanicsLeadScrew := 0.0;
   PRG[29..30].A02_1_PartsCutting.Rollformer.TAxConfig.MechanicsLeadScrew := 622.0;
   PRG[1].A02_1_PartsCutting.Rollformer.TAxConfig.EncoderDistancePerRevolution := 0.0;
   PRG[2..25].A02_1_PartsCutting.Rollformer.TAxConfig.EncoderDistancePerRevolution := 500.0;
   PRG[26].A02_1_PartsCutting.Rollformer.TAxConfig.EncoderDistancePerRevolution := 0.0;
   PRG[27].A02_1_PartsCutting.Rollformer.TAxConfig.EncoderDistancePerRevolution := 500.0;
   PRG[28].A02_1_PartsCutting.Rollformer.TAxConfig.EncoderDistancePerRevolution := 0.0;
   PRG[29..30].A02_1_PartsCutting.Rollformer.TAxConfig.EncoderDistancePerRevolution := 500.0;
   PRG[1].A02_1_PartsCutting.Rollformer.TAxConfig.DynamicsLimitsMaxVelocity := 0.0;
   PRG[2..25].A02_1_PartsCutting.Rollformer.TAxConfig.DynamicsLimitsMaxVelocity := 36000.0;
   PRG[26].A02_1_PartsCutting.Rollformer.TAxConfig.DynamicsLimitsMaxVelocity := 0.0;
   PRG[27].A02_1_PartsCutting.Rollformer.TAxConfig.DynamicsLimitsMaxVelocity := 32000.0;
   PRG[28].A02_1_PartsCutting.Rollformer.TAxConfig.DynamicsLimitsMaxVelocity := 0.0;
   PRG[29..30].A02_1_PartsCutting.Rollformer.TAxConfig.DynamicsLimitsMaxVelocity := 32000.0;
   PRG[1].A02_1_PartsCutting.Rollformer.TAxConfig.DynamicsLimitsVelocity := 0.0;
   PRG[2..25].A02_1_PartsCutting.Rollformer.TAxConfig.DynamicsLimitsVelocity := 36000.0;
   PRG[26].A02_1_PartsCutting.Rollformer.TAxConfig.DynamicsLimitsVelocity := 0.0;
   PRG[27].A02_1_PartsCutting.Rollformer.TAxConfig.DynamicsLimitsVelocity := 30000.0;
   PRG[28].A02_1_PartsCutting.Rollformer.TAxConfig.DynamicsLimitsVelocity := 0.0;
   PRG[29..30].A02_1_PartsCutting.Rollformer.TAxConfig.DynamicsLimitsVelocity := 30000.0;
   PRG[1].A02_1_PartsCutting.Rollformer.TAxConfig.ControlLoop_Kv := 0.0;
   PRG[2..6].A02_1_PartsCutting.Rollformer.TAxConfig.ControlLoop_Kv := 4.0;
   PRG[7].A02_1_PartsCutting.Rollformer.TAxConfig.ControlLoop_Kv := 10.0;
   PRG[8..25].A02_1_PartsCutting.Rollformer.TAxConfig.ControlLoop_Kv := 4.0;
   PRG[26].A02_1_PartsCutting.Rollformer.TAxConfig.ControlLoop_Kv := 0.0;
   PRG[27].A02_1_PartsCutting.Rollformer.TAxConfig.ControlLoop_Kv := 4.0;
   PRG[28].A02_1_PartsCutting.Rollformer.TAxConfig.ControlLoop_Kv := 0.0;
   PRG[29..30].A02_1_PartsCutting.Rollformer.TAxConfig.ControlLoop_Kv := 4.0;
   PRG[1].A02_1_PartsCutting.Rollformer.TAxConfig.ControlLoop_Kpc := 0.0;
   PRG[2..25].A02_1_PartsCutting.Rollformer.TAxConfig.ControlLoop_Kpc := 100.0;
   PRG[26].A02_1_PartsCutting.Rollformer.TAxConfig.ControlLoop_Kpc := 0.0;
   PRG[27].A02_1_PartsCutting.Rollformer.TAxConfig.ControlLoop_Kpc := 100.0;
   PRG[28].A02_1_PartsCutting.Rollformer.TAxConfig.ControlLoop_Kpc := 0.0;
   PRG[29..30].A02_1_PartsCutting.Rollformer.TAxConfig.ControlLoop_Kpc := 100.0;
   PRG[7].A0301_A0302.Trasporto.VelOvr_PLen_UpTo_1000 := 100.0;
   PRG[20].A0301_A0302.Trasporto.VelOvr_PLen_UpTo_1000 := 100.0;
   PRG[23].A0301_A0302.Trasporto.VelOvr_PLen_UpTo_1000 := 100.0;
   PRG[7].A0301_A0302.Trasporto.VelOvr_PLen_UpTo_1500 := 100.0;
   PRG[20].A0301_A0302.Trasporto.VelOvr_PLen_UpTo_1500 := 100.0;
   PRG[23].A0301_A0302.Trasporto.VelOvr_PLen_UpTo_1500 := 100.0;
   PRG[7].A0301_A0302.Trasporto.VelOvr_PLen_UpTo_2000 := 100.0;
   PRG[20].A0301_A0302.Trasporto.VelOvr_PLen_UpTo_2000 := 100.0;
   PRG[23].A0301_A0302.Trasporto.VelOvr_PLen_UpTo_2000 := 100.0;
   PRG[7].A0301_A0302.Trasporto.VelOvr_PLen_UpTo_2500 := 100.0;
   PRG[20].A0301_A0302.Trasporto.VelOvr_PLen_UpTo_2500 := 100.0;
   PRG[23].A0301_A0302.Trasporto.VelOvr_PLen_UpTo_2500 := 100.0;
   PRG[7].A0301_A0302.Trasporto.VelOvr_PLen_UpTo_3000 := 100.0;
   PRG[20].A0301_A0302.Trasporto.VelOvr_PLen_UpTo_3000 := 100.0;
   PRG[23].A0301_A0302.Trasporto.VelOvr_PLen_UpTo_3000 := 100.0;
   PRG[7].A0301_A0302.Trasporto.VelOvr_PLen_UpTo_3500 := 100.0;
   PRG[20].A0301_A0302.Trasporto.VelOvr_PLen_UpTo_3500 := 100.0;
   PRG[23].A0301_A0302.Trasporto.VelOvr_PLen_UpTo_3500 := 100.0;
   PRG[7].A0301_A0302.Trasporto.VelOvr_PLen_UpTo_4000 := 100.0;
   PRG[20].A0301_A0302.Trasporto.VelOvr_PLen_UpTo_4000 := 100.0;
   PRG[23].A0301_A0302.Trasporto.VelOvr_PLen_UpTo_4000 := 100.0;
   PRG[7].A0301_A0302.Trasporto.VelOvr_PLen_UpTo_4500 := 100.0;
   PRG[20].A0301_A0302.Trasporto.VelOvr_PLen_UpTo_4500 := 100.0;
   PRG[23].A0301_A0302.Trasporto.VelOvr_PLen_UpTo_4500 := 100.0;
   PRG[7].A0301_A0302.Trasporto.VelOvr_PLen_UpTo_5000 := 100.0;
   PRG[20].A0301_A0302.Trasporto.VelOvr_PLen_UpTo_5000 := 100.0;
   PRG[23].A0301_A0302.Trasporto.VelOvr_PLen_UpTo_5000 := 100.0;
   PRG[7].A0301_A0302.Trasporto.VelOvr_PLen_UpTo_5500 := 100.0;
   PRG[20].A0301_A0302.Trasporto.VelOvr_PLen_UpTo_5500 := 100.0;
   PRG[23].A0301_A0302.Trasporto.VelOvr_PLen_UpTo_5500 := 100.0;
   PRG[7].A0301_A0302.Ribaltatore.VelOvr_PLen_UpTo_1000 := 100.0;
   PRG[20].A0301_A0302.Ribaltatore.VelOvr_PLen_UpTo_1000 := 100.0;
   PRG[23].A0301_A0302.Ribaltatore.VelOvr_PLen_UpTo_1000 := 100.0;
   PRG[7].A0301_A0302.Ribaltatore.VelOvr_PLen_UpTo_1500 := 100.0;
   PRG[20].A0301_A0302.Ribaltatore.VelOvr_PLen_UpTo_1500 := 100.0;
   PRG[23].A0301_A0302.Ribaltatore.VelOvr_PLen_UpTo_1500 := 100.0;
   PRG[7].A0301_A0302.Ribaltatore.VelOvr_PLen_UpTo_2000 := 100.0;
   PRG[20].A0301_A0302.Ribaltatore.VelOvr_PLen_UpTo_2000 := 100.0;
   PRG[23].A0301_A0302.Ribaltatore.VelOvr_PLen_UpTo_2000 := 100.0;
   PRG[7].A0301_A0302.Ribaltatore.VelOvr_PLen_UpTo_2500 := 100.0;
   PRG[20].A0301_A0302.Ribaltatore.VelOvr_PLen_UpTo_2500 := 100.0;
   PRG[23].A0301_A0302.Ribaltatore.VelOvr_PLen_UpTo_2500 := 100.0;
   PRG[7].A0301_A0302.Ribaltatore.VelOvr_PLen_UpTo_3000 := 100.0;
   PRG[20].A0301_A0302.Ribaltatore.VelOvr_PLen_UpTo_3000 := 100.0;
   PRG[23].A0301_A0302.Ribaltatore.VelOvr_PLen_UpTo_3000 := 100.0;
   PRG[7].A0301_A0302.Ribaltatore.VelOvr_PLen_UpTo_3500 := 100.0;
   PRG[20].A0301_A0302.Ribaltatore.VelOvr_PLen_UpTo_3500 := 100.0;
   PRG[23].A0301_A0302.Ribaltatore.VelOvr_PLen_UpTo_3500 := 100.0;
   PRG[7].A0301_A0302.Ribaltatore.VelOvr_PLen_UpTo_4000 := 100.0;
   PRG[20].A0301_A0302.Ribaltatore.VelOvr_PLen_UpTo_4000 := 100.0;
   PRG[23].A0301_A0302.Ribaltatore.VelOvr_PLen_UpTo_4000 := 100.0;
   PRG[7].A0301_A0302.Ribaltatore.VelOvr_PLen_UpTo_4500 := 100.0;
   PRG[20].A0301_A0302.Ribaltatore.VelOvr_PLen_UpTo_4500 := 100.0;
   PRG[23].A0301_A0302.Ribaltatore.VelOvr_PLen_UpTo_4500 := 100.0;
   PRG[7].A0301_A0302.Ribaltatore.VelOvr_PLen_UpTo_5000 := 100.0;
   PRG[20].A0301_A0302.Ribaltatore.VelOvr_PLen_UpTo_5000 := 100.0;
   PRG[23].A0301_A0302.Ribaltatore.VelOvr_PLen_UpTo_5000 := 100.0;
   PRG[7].A0301_A0302.Ribaltatore.VelOvr_PLen_UpTo_5500 := 100.0;
   PRG[20].A0301_A0302.Ribaltatore.VelOvr_PLen_UpTo_5500 := 100.0;
   PRG[23].A0301_A0302.Ribaltatore.VelOvr_PLen_UpTo_5500 := 100.0;
   PRG[7].A0301_A0302.Ribaltatore.Pos_1_Delay := T#1S;
   PRG[20].A0301_A0302.Ribaltatore.Pos_1_Delay := T#1S;
   PRG[23].A0301_A0302.Ribaltatore.Pos_1_Delay := T#1S;
   PRG[7].A0301_A0302.Bordatrice.VelOvr_PLen_UpTo_1000 := 100.0;
   PRG[20].A0301_A0302.Bordatrice.VelOvr_PLen_UpTo_1000 := 100.0;
   PRG[23].A0301_A0302.Bordatrice.VelOvr_PLen_UpTo_1000 := 100.0;
   PRG[7].A0301_A0302.Bordatrice.VelOvr_PLen_UpTo_1500 := 100.0;
   PRG[20].A0301_A0302.Bordatrice.VelOvr_PLen_UpTo_1500 := 100.0;
   PRG[23].A0301_A0302.Bordatrice.VelOvr_PLen_UpTo_1500 := 100.0;
   PRG[7].A0301_A0302.Bordatrice.VelOvr_PLen_UpTo_2000 := 100.0;
   PRG[20].A0301_A0302.Bordatrice.VelOvr_PLen_UpTo_2000 := 100.0;
   PRG[23].A0301_A0302.Bordatrice.VelOvr_PLen_UpTo_2000 := 100.0;
   PRG[7].A0301_A0302.Bordatrice.VelOvr_PLen_UpTo_2500 := 100.0;
   PRG[20].A0301_A0302.Bordatrice.VelOvr_PLen_UpTo_2500 := 100.0;
   PRG[23].A0301_A0302.Bordatrice.VelOvr_PLen_UpTo_2500 := 100.0;
   PRG[7].A0301_A0302.Bordatrice.VelOvr_PLen_UpTo_3000 := 100.0;
   PRG[20].A0301_A0302.Bordatrice.VelOvr_PLen_UpTo_3000 := 100.0;
   PRG[23].A0301_A0302.Bordatrice.VelOvr_PLen_UpTo_3000 := 100.0;
   PRG[7].A0301_A0302.Bordatrice.VelOvr_PLen_UpTo_3500 := 100.0;
   PRG[20].A0301_A0302.Bordatrice.VelOvr_PLen_UpTo_3500 := 100.0;
   PRG[23].A0301_A0302.Bordatrice.VelOvr_PLen_UpTo_3500 := 100.0;
   PRG[7].A0301_A0302.Bordatrice.VelOvr_PLen_UpTo_4000 := 100.0;
   PRG[20].A0301_A0302.Bordatrice.VelOvr_PLen_UpTo_4000 := 100.0;
   PRG[23].A0301_A0302.Bordatrice.VelOvr_PLen_UpTo_4000 := 100.0;
   PRG[7].A0301_A0302.Bordatrice.VelOvr_PLen_UpTo_4500 := 100.0;
   PRG[20].A0301_A0302.Bordatrice.VelOvr_PLen_UpTo_4500 := 100.0;
   PRG[23].A0301_A0302.Bordatrice.VelOvr_PLen_UpTo_4500 := 100.0;
   PRG[7].A0301_A0302.Bordatrice.VelOvr_PLen_UpTo_5000 := 100.0;
   PRG[20].A0301_A0302.Bordatrice.VelOvr_PLen_UpTo_5000 := 100.0;
   PRG[23].A0301_A0302.Bordatrice.VelOvr_PLen_UpTo_5000 := 100.0;
   PRG[7].A0301_A0302.Bordatrice.VelOvr_PLen_UpTo_5500 := 100.0;
   PRG[20].A0301_A0302.Bordatrice.VelOvr_PLen_UpTo_5500 := 100.0;
   PRG[23].A0301_A0302.Bordatrice.VelOvr_PLen_UpTo_5500 := 100.0;
   PRG[7].A0303_A0304.Trasporto.VelOvr_PLen_UpTo_1000 := 100.0;
   PRG[20].A0303_A0304.Trasporto.VelOvr_PLen_UpTo_1000 := 100.0;
   PRG[23].A0303_A0304.Trasporto.VelOvr_PLen_UpTo_1000 := 100.0;
   PRG[7].A0303_A0304.Trasporto.VelOvr_PLen_UpTo_1500 := 100.0;
   PRG[20].A0303_A0304.Trasporto.VelOvr_PLen_UpTo_1500 := 100.0;
   PRG[23].A0303_A0304.Trasporto.VelOvr_PLen_UpTo_1500 := 100.0;
   PRG[7].A0303_A0304.Trasporto.VelOvr_PLen_UpTo_2000 := 100.0;
   PRG[20].A0303_A0304.Trasporto.VelOvr_PLen_UpTo_2000 := 100.0;
   PRG[23].A0303_A0304.Trasporto.VelOvr_PLen_UpTo_2000 := 100.0;
   PRG[7].A0303_A0304.Trasporto.VelOvr_PLen_UpTo_2500 := 100.0;
   PRG[20].A0303_A0304.Trasporto.VelOvr_PLen_UpTo_2500 := 100.0;
   PRG[23].A0303_A0304.Trasporto.VelOvr_PLen_UpTo_2500 := 100.0;
   PRG[7].A0303_A0304.Trasporto.VelOvr_PLen_UpTo_3000 := 100.0;
   PRG[20].A0303_A0304.Trasporto.VelOvr_PLen_UpTo_3000 := 100.0;
   PRG[23].A0303_A0304.Trasporto.VelOvr_PLen_UpTo_3000 := 100.0;
   PRG[7].A0303_A0304.Trasporto.VelOvr_PLen_UpTo_3500 := 100.0;
   PRG[20].A0303_A0304.Trasporto.VelOvr_PLen_UpTo_3500 := 100.0;
   PRG[23].A0303_A0304.Trasporto.VelOvr_PLen_UpTo_3500 := 100.0;
   PRG[7].A0303_A0304.Trasporto.VelOvr_PLen_UpTo_4000 := 100.0;
   PRG[20].A0303_A0304.Trasporto.VelOvr_PLen_UpTo_4000 := 100.0;
   PRG[23].A0303_A0304.Trasporto.VelOvr_PLen_UpTo_4000 := 100.0;
   PRG[7].A0303_A0304.Trasporto.VelOvr_PLen_UpTo_4500 := 100.0;
   PRG[20].A0303_A0304.Trasporto.VelOvr_PLen_UpTo_4500 := 100.0;
   PRG[23].A0303_A0304.Trasporto.VelOvr_PLen_UpTo_4500 := 100.0;
   PRG[7].A0303_A0304.Trasporto.VelOvr_PLen_UpTo_5000 := 100.0;
   PRG[20].A0303_A0304.Trasporto.VelOvr_PLen_UpTo_5000 := 100.0;
   PRG[23].A0303_A0304.Trasporto.VelOvr_PLen_UpTo_5000 := 100.0;
   PRG[7].A0303_A0304.Trasporto.VelOvr_PLen_UpTo_5500 := 100.0;
   PRG[20].A0303_A0304.Trasporto.VelOvr_PLen_UpTo_5500 := 100.0;
   PRG[23].A0303_A0304.Trasporto.VelOvr_PLen_UpTo_5500 := 100.0;
   PRG[7].A0303_A0304.Navetta.VelOvr_PLen_UpTo_1000 := 100.0;
   PRG[20].A0303_A0304.Navetta.VelOvr_PLen_UpTo_1000 := 100.0;
   PRG[23].A0303_A0304.Navetta.VelOvr_PLen_UpTo_1000 := 100.0;
   PRG[7].A0303_A0304.Navetta.VelOvr_PLen_UpTo_1500 := 100.0;
   PRG[20].A0303_A0304.Navetta.VelOvr_PLen_UpTo_1500 := 100.0;
   PRG[23].A0303_A0304.Navetta.VelOvr_PLen_UpTo_1500 := 100.0;
   PRG[7].A0303_A0304.Navetta.VelOvr_PLen_UpTo_2000 := 100.0;
   PRG[20].A0303_A0304.Navetta.VelOvr_PLen_UpTo_2000 := 100.0;
   PRG[23].A0303_A0304.Navetta.VelOvr_PLen_UpTo_2000 := 100.0;
   PRG[7].A0303_A0304.Navetta.VelOvr_PLen_UpTo_2500 := 100.0;
   PRG[20].A0303_A0304.Navetta.VelOvr_PLen_UpTo_2500 := 100.0;
   PRG[23].A0303_A0304.Navetta.VelOvr_PLen_UpTo_2500 := 100.0;
   PRG[7].A0303_A0304.Navetta.VelOvr_PLen_UpTo_3000 := 100.0;
   PRG[20].A0303_A0304.Navetta.VelOvr_PLen_UpTo_3000 := 100.0;
   PRG[23].A0303_A0304.Navetta.VelOvr_PLen_UpTo_3000 := 100.0;
   PRG[7].A0303_A0304.Navetta.VelOvr_PLen_UpTo_3500 := 100.0;
   PRG[20].A0303_A0304.Navetta.VelOvr_PLen_UpTo_3500 := 100.0;
   PRG[23].A0303_A0304.Navetta.VelOvr_PLen_UpTo_3500 := 100.0;
   PRG[7].A0303_A0304.Navetta.VelOvr_PLen_UpTo_4000 := 100.0;
   PRG[20].A0303_A0304.Navetta.VelOvr_PLen_UpTo_4000 := 100.0;
   PRG[23].A0303_A0304.Navetta.VelOvr_PLen_UpTo_4000 := 100.0;
   PRG[7].A0303_A0304.Navetta.VelOvr_PLen_UpTo_4500 := 100.0;
   PRG[20].A0303_A0304.Navetta.VelOvr_PLen_UpTo_4500 := 100.0;
   PRG[23].A0303_A0304.Navetta.VelOvr_PLen_UpTo_4500 := 100.0;
   PRG[7].A0303_A0304.Navetta.VelOvr_PLen_UpTo_5000 := 100.0;
   PRG[20].A0303_A0304.Navetta.VelOvr_PLen_UpTo_5000 := 100.0;
   PRG[23].A0303_A0304.Navetta.VelOvr_PLen_UpTo_5000 := 100.0;
   PRG[7].A0303_A0304.Navetta.VelOvr_PLen_UpTo_5500 := 100.0;
   PRG[20].A0303_A0304.Navetta.VelOvr_PLen_UpTo_5500 := 100.0;
   PRG[23].A0303_A0304.Navetta.VelOvr_PLen_UpTo_5500 := 100.0;
END_DATA_BLOCK
